FUNCTION_BLOCK FB_JoyInputScale
VAR_INPUT
	nJoyX : INT := G_Inputs.nCylPos;
	bIsManual : BOOL;
	stJoyInputScale : ST_JoyInputScale; 
END_VAR

VAR_OUTPUT
	fJoyX_Norm : LREAL;
END_VAR

VAR
	fRawInput : LREAL;
	fTempInput : LREAL;
	fTempOutput : LREAL;
END_VAR

fRawInput := INT_TO_REAL(nJoyX);

fTempInput := fRawInput - stJoyInputScale.fNeutralInputVal; 

IF fTempInput > stJoyInputScale.fNeutralDeadband THEN
	fTempOutput := fTempInput/(stJoyInputScale.fMaxInputVal - stJoyInputScale.fNeutralInputVal); 

ELSIF fTempInput < -stJoyInputScale.fNeutralDeadband THEN
	fTempOutput := fTempInput/(stJoyInputScale.fNeutralInputVal - stJoyInputScale.fMinInputVal);
	
ELSE
	fTempOutput := 0.0; 
END_IF

IF NOT(bIsManual) THEN
	fJoyX_Norm := 0.0;
ELSE
	fJoyX_Norm := LIMIT(stJoyInputScale.fMinOutputValue, fTempOutput, stJoyInputScale.fMaxOutputValue); 
END_IF

END_FUNCTION_BLOCK

(* stored: Version 1.1.0.1, ProductVersion 3.1.4024.12
   POU FB_JoyInputScale: Id {1a744545-8e9f-42d2-9c5e-33b2dfe99fe9}, SpecialFunc None *)
